Omron CX-Programmer project NewProject (CX-Programmer 9.75)

# PLC SCADAPTG: CP2E-N N

## Global symbols (name address type ; comment)
100.01 BOOL  ; CIO
100.03 BOOL  ; CIO
A401 CHANNEL  ; CP1W-ADB21 PT100 Analog Input Option Board
D1024 CHANNEL  ; Data Register
inst_ModbusServer _CP2E003_ExecuteModTcpServer
inst_SCADA SCADA_Control_FB

## Program SCADAPTG (cyclic task 0)
Local symbols
M1_DirEdge1 W2.05 BOOL
M1_DirEdge2 W2.06 BOOL
M1_Stopping W2.07 BOOL
M2_DirEdge1 W3.00 BOOL
M2_DirEdge2 W3.01 BOOL
M2_Stopping W3.02 BOOL

### Section SCADA_Control

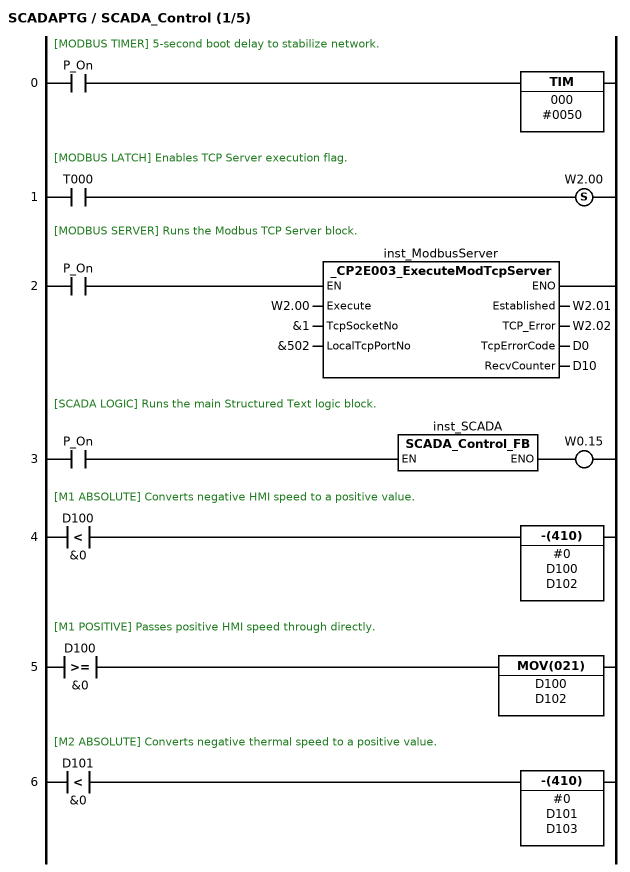
; rung 0: [MODBUS TIMER] 5-second boot delay to stabilize network.
LD P_On
TIM 000 #0050
; rung 1: [MODBUS LATCH] Enables TCP Server execution flag.
LD T000
SET W2.00
; rung 2: [MODBUS SERVER] Runs the Modbus TCP Server block.
LD P_On
CALL inst_ModbusServer : _CP2E003_ExecuteModTcpServer (Execute := W2.00, TcpSocketNo := &1, LocalTcpPortNo := &502, Established => W2.01, TCP_Error => W2.02, TcpErrorCode => D0, RecvCounter => D10)
; rung 3: [SCADA LOGIC] Runs the main Structured Text logic block.
LD P_On
CALL inst_SCADA : SCADA_Control_FB ()
OUT W0.15
; rung 4: [M1 ABSOLUTE] Converts negative HMI speed to a positive value.
LD<S(312) D100 &0
-(410) #0 D100 D102
; rung 5: [M1 POSITIVE] Passes positive HMI speed through directly.
LD>=S(327) D100 &0
MOV(021) D100 D102
; rung 6: [M2 ABSOLUTE] Converts negative thermal speed to a positive value.
LD<S(312) D101 &0
-(410) #0 D101 D103

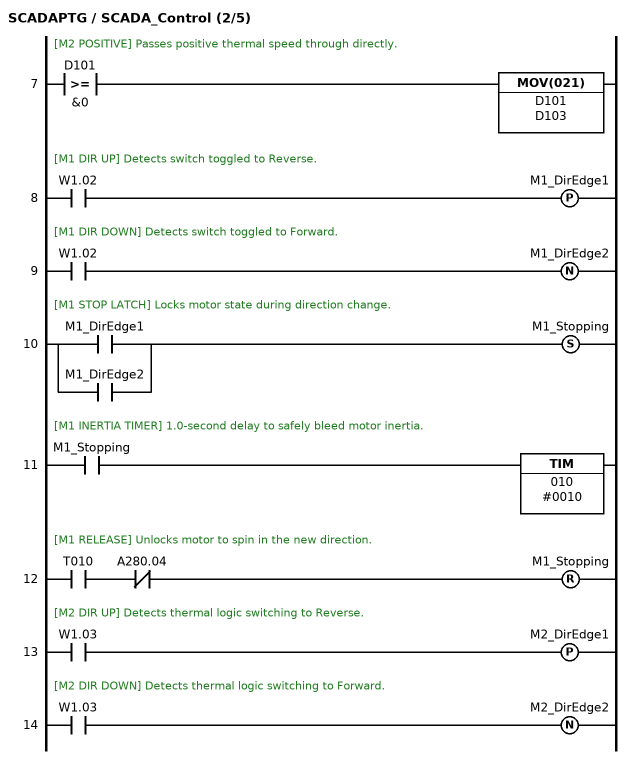
; rung 7: [M2 POSITIVE] Passes positive thermal speed through directly.
LD>=S(327) D101 &0
MOV(021) D101 D103
; rung 8: [M1 DIR UP] Detects switch toggled to Reverse.
LD W1.02
DIFU(013) M1_DirEdge1
; rung 9: [M1 DIR DOWN] Detects switch toggled to Forward.
LD W1.02
DIFD(014) M1_DirEdge2
; rung 10: [M1 STOP LATCH] Locks motor state during direction change.
LD M1_DirEdge1
OR M1_DirEdge2
SET M1_Stopping
; rung 11: [M1 INERTIA TIMER] 1.0-second delay to safely bleed motor inertia.
LD M1_Stopping
TIM 010 #0010
; rung 12: [M1 RELEASE] Unlocks motor to spin in the new direction.
LD T010
ANDNOT A280.04
RSET M1_Stopping
; rung 13: [M2 DIR UP] Detects thermal logic switching to Reverse.
LD W1.03
DIFU(013) M2_DirEdge1
; rung 14: [M2 DIR DOWN] Detects thermal logic switching to Forward.
LD W1.03
DIFD(014) M2_DirEdge2

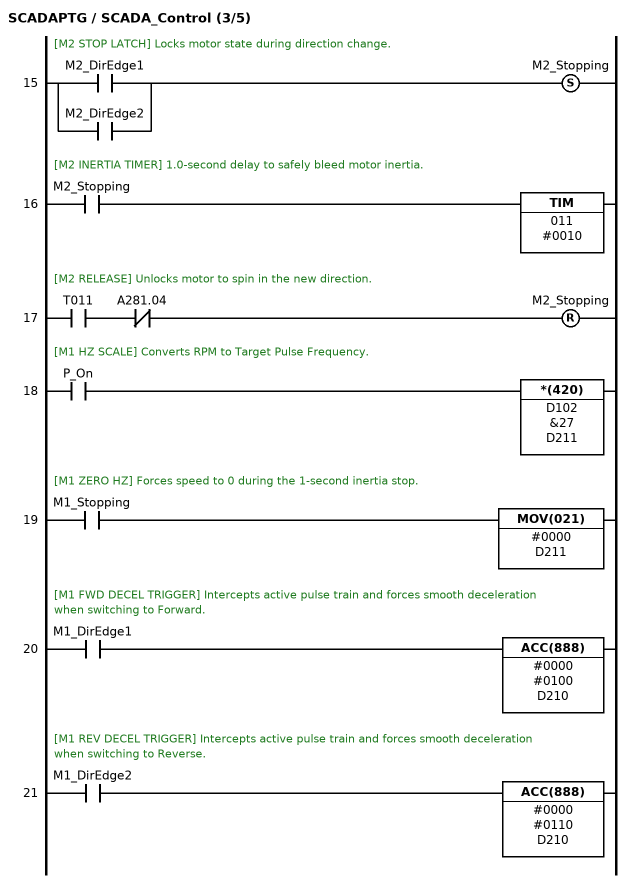
; rung 15: [M2 STOP LATCH] Locks motor state during direction change.
LD M2_DirEdge1
OR M2_DirEdge2
SET M2_Stopping
; rung 16: [M2 INERTIA TIMER] 1.0-second delay to safely bleed motor inertia.
LD M2_Stopping
TIM 011 #0010
; rung 17: [M2 RELEASE] Unlocks motor to spin in the new direction.
LD T011
ANDNOT A281.04
RSET M2_Stopping
; rung 18: [M1 HZ SCALE] Converts RPM to Target Pulse Frequency.
LD P_On
*(420) D102 &27 D211
; rung 19: [M1 ZERO HZ] Forces speed to 0 during the 1-second inertia stop.
LD M1_Stopping
MOV(021) #0000 D211
; rung 20: [M1 FWD DECEL TRIGGER] Intercepts active pulse train and forces smooth deceleration when switching to Forward.
LD M1_DirEdge1
ACC(888) #0000 #0100 D210
; rung 21: [M1 REV DECEL TRIGGER] Intercepts active pulse train and forces smooth deceleration when switching to Reverse.
LD M1_DirEdge2
ACC(888) #0000 #0110 D210

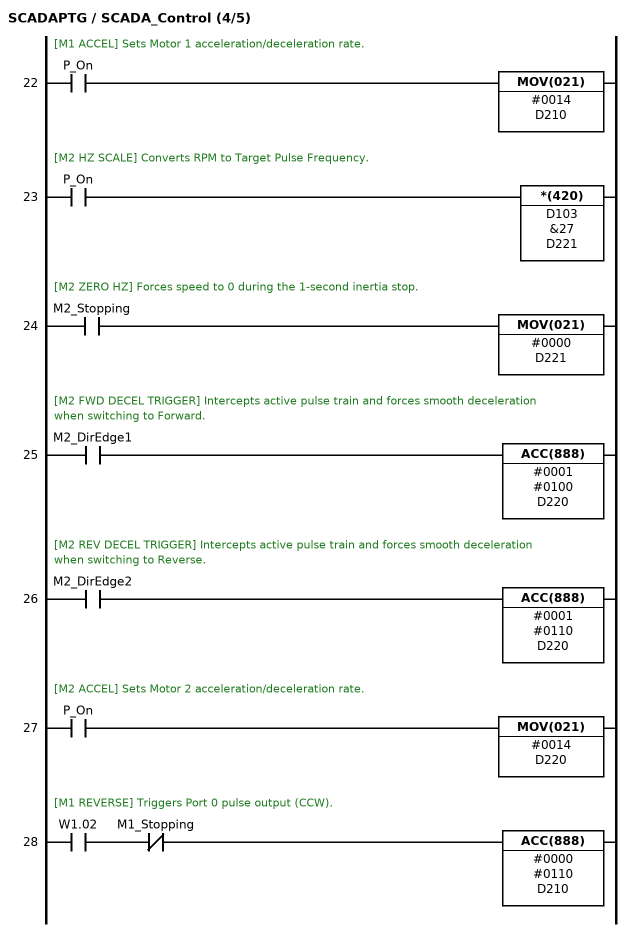
; rung 22: [M1 ACCEL] Sets Motor 1 acceleration/deceleration rate.
LD P_On
MOV(021) #0014 D210
; rung 23: [M2 HZ SCALE] Converts RPM to Target Pulse Frequency.
LD P_On
*(420) D103 &27 D221
; rung 24: [M2 ZERO HZ] Forces speed to 0 during the 1-second inertia stop.
LD M2_Stopping
MOV(021) #0000 D221
; rung 25: [M2 FWD DECEL TRIGGER] Intercepts active pulse train and forces smooth deceleration when switching to Forward.
LD M2_DirEdge1
ACC(888) #0001 #0100 D220
; rung 26: [M2 REV DECEL TRIGGER] Intercepts active pulse train and forces smooth deceleration when switching to Reverse.
LD M2_DirEdge2
ACC(888) #0001 #0110 D220
; rung 27: [M2 ACCEL] Sets Motor 2 acceleration/deceleration rate.
LD P_On
MOV(021) #0014 D220
; rung 28: [M1 REVERSE] Triggers Port 0 pulse output (CCW).
LD W1.02
ANDNOT M1_Stopping
ACC(888) #0000 #0110 D210

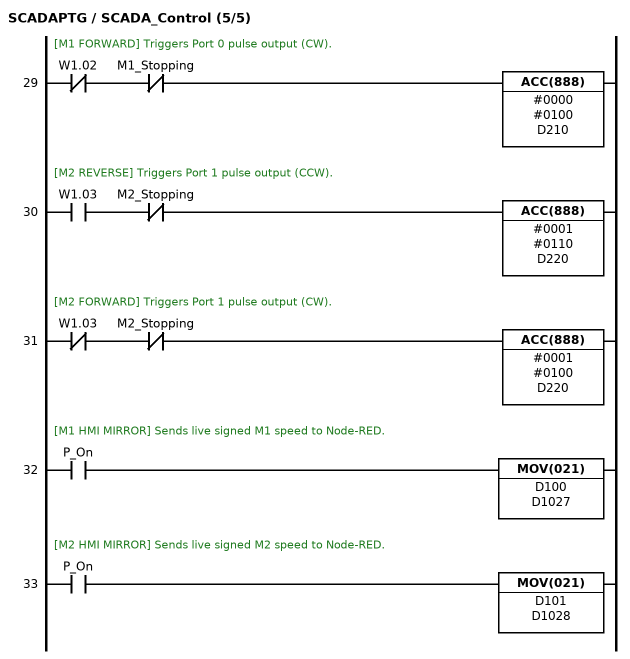
; rung 29: [M1 FORWARD] Triggers Port 0 pulse output (CW).
LDNOT W1.02
ANDNOT M1_Stopping
ACC(888) #0000 #0100 D210
; rung 30: [M2 REVERSE] Triggers Port 1 pulse output (CCW).
LD W1.03
ANDNOT M2_Stopping
ACC(888) #0001 #0110 D220
; rung 31: [M2 FORWARD] Triggers Port 1 pulse output (CW).
LDNOT W1.03
ANDNOT M2_Stopping
ACC(888) #0001 #0100 D220
; rung 32: [M1 HMI MIRROR] Sends live signed M1 speed to Node-RED.
LD P_On
MOV(021) D100 D1027
; rung 33: [M2 HMI MIRROR] Sends live signed M2 speed to Node-RED.
LD P_On
MOV(021) D101 D1028

### Section END
; rung 0
END(001)

## Function block _CP2E003_ExecuteModTcpServer (Omron library block, body left out)

## Function block SCADA_Control_FB
VAR
  Field_Motor1_Button AT 0.00 : BOOL;  (* Field Motor 1 Enable Toggle (NO) *)
  Field_E_Stop AT 0.01 : BOOL;  (* Field Emergency Button *)
  Field_Reset_Button AT 0.02 : BOOL;  (* Field Safety Reset (NC) *)
  Field_Motor2_Button AT 0.03 : BOOL;  (* Field Motor 2 Enable Toggle (NO) *)
  Field_E_Stop_Status AT W0.03 : BOOL;  (* XB2BS42C Emergency Button Status *)
  Edge_Storage AT W0.00 : BOOL;  (* One-shot memory bit for edge detection *)
  HMI_E_Stop AT W0.01 : BOOL;  (* Modbus Coil 1 (Node-RED Emergency Stop) *)
  HMI_Reset AT W0.02 : BOOL;  (* Modbus Coil 2 (Node-RED Safety Reset) *)
  Safety_Latch AT W0.04 : BOOL;  (* Master Safety Lockout Latch Bit *)
  Motor1_Status AT W0.05 : BOOL;  (* Modbus Coil 5 (Node-RED Motor 1 LED) *)
  Motor2_Status AT W0.06 : BOOL;  (* Modbus Coil 6 (Node-RED Motor 2 LED) *)
  HMI_Button AT W0.07 : BOOL;  (* Modbus Coil 7 (Node-RED Field Override Badge) *)
  HMI_Motor1_Enable AT W1.00 : BOOL;  (* Modbus Coil 8 (Node-RED Motor 1 Switch) *)
  HMI_Motor2_Enable AT W1.01 : BOOL;  (* Modbus Coil 9 (Node-RED Motor 2 Switch) *)
  HMI_Motor1_Dir AT W1.02 : BOOL;  (* Modbus Coil 10 (Node-RED Motor 1 Direction) *)
  HMI_Motor2_Dir AT W1.03 : BOOL;  (* Modbus Coil 11 (Node-RED Motor 2 Direction) *)
  Motor1_Speed AT D100 : INT;  (* Speed Command to TB6600 Driver #1 *)
  Motor2_Speed AT D101 : INT;  (* Speed Command to TB6600 Driver #2 *)
  Raw_Temp AT D1024 : INT;  (* CP1W-ADB21 Analog In (PT100 Temp x100) *)
  Raw_Temp_Input AT 80 : INT;  (* Raw data of PT100 Temp *)
  HMI_Motor1_Cmd AT D1025 : INT;  (* Node-RED Speed Slider Command *)
  HMI_Motor2_Cmd AT D1026 : INT;  (* Calculated Thermal Auto-Speed (Preview RPM) *)
  Motor2_Edge_Storage : BOOL;  (* One-shot memory bit for Motor 2 field toggle *)
  HMI_Motor2_Button : BOOL;  (* Field override state for Motor 2 *)
END_VAR
 (* 1. DUAL SAFETY LATCH LOGIC (Physical E-Stop + HMI E-Stop + Field Reset)   *)
(* System is safe ONLY if HMI E-Stop is OFF AND Field E-Stop button is healthy *)
Safety_Latch := NOT(HMI_E_Stop) AND Field_E_Stop AND (HMI_Reset OR NOT(Field_Reset_Button) OR Safety_Latch);

(* 2. FIELD BUTTON TOGGLE - MOTOR 1 (Edge Detection + Flip-Flop)             *)
IF Field_Motor1_Button AND NOT Edge_Storage THEN
    HMI_Button := NOT HMI_Button; (* Toggle Field Override State *)
END_IF;
Edge_Storage := Field_Motor1_Button; (* Save state for edge detection *)

(* 2b. FIELD BUTTON TOGGLE - MOTOR 2 (Edge Detection + Flip-Flop)            *)
IF Field_Motor2_Button AND NOT Motor2_Edge_Storage THEN
    HMI_Motor2_Button := NOT HMI_Motor2_Button; (* Toggle Field Override State for Motor 2 *)
END_IF;
Motor2_Edge_Storage := Field_Motor2_Button; (* Save state for edge detection *)

(* 3. TEMPERATURE SENSOR SCALING (0-100C Range) *)
(* Transmitter is 0-10V linear output, calibrated directly to 0-100C.       *)
(* CP1W-ADB21 voltage input gives 0-4000 counts across 0-10V.               *)
(* Raw_Temp is stored x100, so: Temp(x100) = Raw_Temp_Input * 100 / 40      *)
IF Raw_Temp_Input <= 0 THEN
    Raw_Temp := 0; (* Prevent negative numbers on wire break or noise *)
ELSE
    Raw_Temp := (Raw_Temp_Input * 5) / 2;
END_IF;

(* Automated Thermal Speed Logic based on 0-100C Scale *)
IF Raw_Temp <= 3000 THEN          (* below 30.00ｰC *)
    HMI_Motor2_Cmd := 25;         (* floor: 25 RPM *)
ELSIF Raw_Temp >= 6000 THEN       (* above 60.00ｰC *)
    HMI_Motor2_Cmd := 500;        (* ceiling: 500 RPM *)
ELSE
    HMI_Motor2_Cmd := 25 + DINT_TO_INT((INT_TO_DINT(Raw_Temp - 3000) * 19) / 120);
END_IF;

(* 4. MASTER SAFETY INTERLOCK & MOTOR SPEED EVALUATION                       *)
IF NOT Safety_Latch THEN
    (* EMERGENCY STOP ACTIVE: Drop all speeds to 0 immediately *)
    Motor1_Speed := 0;
    Motor2_Speed := 0;
    HMI_Button := FALSE; (* Reset field toggle bit *)
    HMI_Motor2_Button := FALSE; (* Reset Motor 2 field toggle bit *)
ELSE
    (* SYSTEM SAFE: Evaluate individual motor channels *)
    (* --- MOTOR 1: Manual HMI Channel --- *)
    IF (HMI_Motor1_Enable OR HMI_Button) THEN
        IF HMI_Motor1_Dir THEN
            Motor1_Speed := ABS(HMI_Motor1_Cmd) * -1; (* Reverse *)
        ELSE
            Motor1_Speed := ABS(HMI_Motor1_Cmd);      (* Forward *)
        END_IF;
    ELSE
        Motor1_Speed := 0;
    END_IF;
    (* --- MOTOR 2: Automated Thermal Channel --- *)
    IF (HMI_Motor2_Enable OR HMI_Motor2_Button) THEN
        IF HMI_Motor2_Dir THEN
            Motor2_Speed := HMI_Motor2_Cmd * -1; (* Reverse *)
        ELSE
            Motor2_Speed := HMI_Motor2_Cmd;      (* Forward *)
        END_IF;
    ELSE
        Motor2_Speed := 0;
    END_IF;
END_IF;

(* 5. UPDATE MOTOR RUNNING STATUS & PHYSICAL E-STOP BADGES FOR NODE-RED *)
Motor1_Status := (Motor1_Speed <> 0);
Motor2_Status := (Motor2_Speed <> 0);
(* Mirror Physical Field E-Stop hardware pin status to Modbus Coil 3 *)
Field_E_Stop_Status := Field_E_Stop;